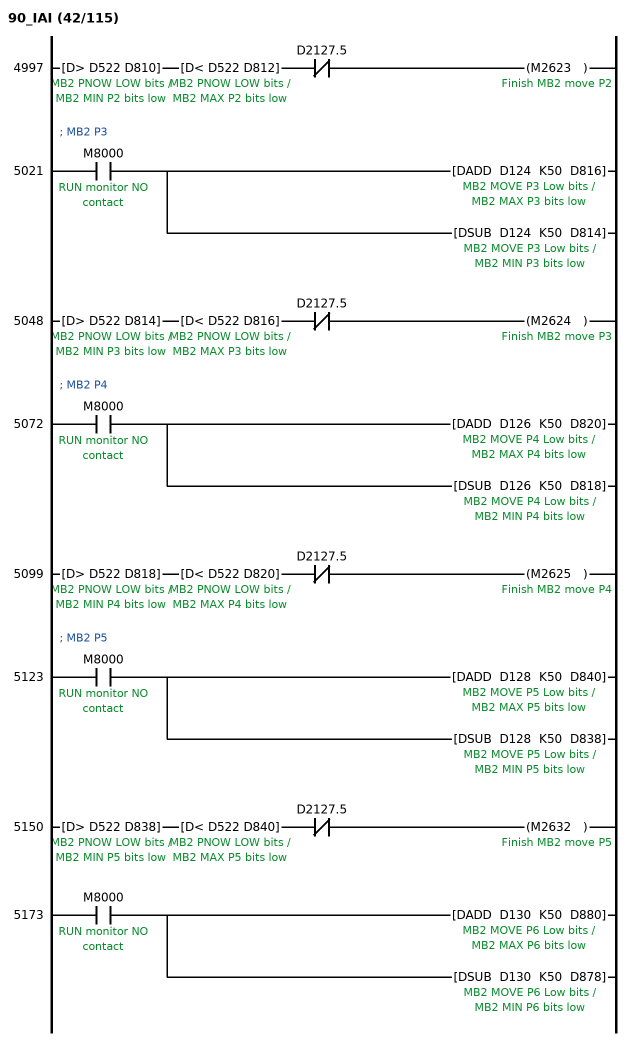
[picture p144: ladder of 90_IAI, rungs at steps 4997 to 5173]
4997  LDD>    D522 D810  ; MB2 PNOW LOW bits / MB2 MIN P2 bits low
      ANDD<   D522 D812  ; MB2 PNOW LOW bits / MB2 MAX P2 bits low
      ANI     D2127.5
      OUT     M2623  ; Finish MB2 move P2
; MB2 P3
5021  LD      M8000  ; RUN monitor NO contact
      DADD    D124 K50 D816  ; MB2 MAX P3 bits low
      DSUB    D124 K50 D814  ; MB2 MIN P3 bits low
5048  LDD>    D522 D814  ; MB2 PNOW LOW bits / MB2 MIN P3 bits low
      ANDD<   D522 D816  ; MB2 PNOW LOW bits / MB2 MAX P3 bits low
      ANI     D2127.5
      OUT     M2624  ; Finish MB2 move P3
; MB2 P4
5072  LD      M8000  ; RUN monitor NO contact
      DADD    D126 K50 D820  ; MB2 MAX P4 bits low
      DSUB    D126 K50 D818  ; MB2 MIN P4 bits low
5099  LDD>    D522 D818  ; MB2 PNOW LOW bits / MB2 MIN P4 bits low
      ANDD<   D522 D820  ; MB2 PNOW LOW bits / MB2 MAX P4 bits low
      ANI     D2127.5
      OUT     M2625  ; Finish MB2 move P4
; MB2 P5
5123  LD      M8000  ; RUN monitor NO contact
      DADD    D128 K50 D840  ; MB2 MAX P5 bits low
      DSUB    D128 K50 D838  ; MB2 MIN P5 bits low
5150  LDD>    D522 D838  ; MB2 PNOW LOW bits / MB2 MIN P5 bits low
      ANDD<   D522 D840  ; MB2 PNOW LOW bits / MB2 MAX P5 bits low
      ANI     D2127.5
      OUT     M2632  ; Finish MB2 move P5
5173  LD      M8000  ; RUN monitor NO contact
      DADD    D130 K50 D880  ; MB2 MAX P6 bits low
      DSUB    D130 K50 D878  ; MB2 MIN P6 bits low
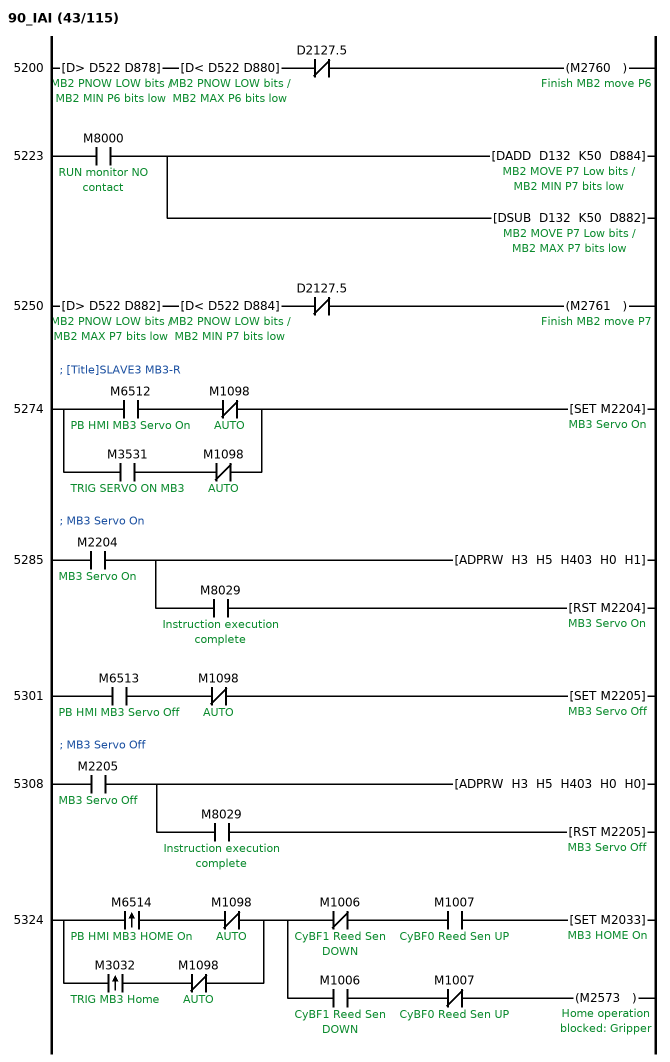
5200  LDD>    D522 D878  ; MB2 PNOW LOW bits / MB2 MIN P6 bits low
      ANDD<   D522 D880  ; MB2 PNOW LOW bits / MB2 MAX P6 bits low
      ANI     D2127.5
      OUT     M2760  ; Finish MB2 move P6
5223  LD      M8000  ; RUN monitor NO contact
      DADD    D132 K50 D884  ; MB2 MIN P7 bits low
      DSUB    D132 K50 D882  ; MB2 MAX P7 bits low
5250  LDD>    D522 D882  ; MB2 PNOW LOW bits / MB2 MAX P7 bits low
      ANDD<   D522 D884  ; MB2 PNOW LOW bits / MB2 MIN P7 bits low
      ANI     D2127.5
      OUT     M2761  ; Finish MB2 move P7
; [Title]SLAVE3 MB3-R
5274  LD      M6512  ; PB HMI MB3 Servo On
      ANI     M1098  ; AUTO
      LD      M3531  ; TRIG SERVO ON MB3
      ANI     M1098  ; AUTO
      ORB
      SET     M2204  ; MB3 Servo On
; MB3 Servo On
5285  LD      M2204  ; MB3 Servo On
      ADPRW   H3 H5 H403 H0 H1
      AND     M8029  ; Instruction execution complete
      RST     M2204  ; MB3 Servo On
5301  LD      M6513  ; PB HMI MB3 Servo Off
      ANI     M1098  ; AUTO
      SET     M2205  ; MB3 Servo Off
; MB3 Servo Off
5308  LD      M2205  ; MB3 Servo Off
      ADPRW   H3 H5 H403 H0 H0
      AND     M8029  ; Instruction execution complete
      RST     M2205  ; MB3 Servo Off
5324  LDP     M6514  ; PB HMI MB3 HOME On
      ANI     M1098  ; AUTO
      LDP     M3032  ; TRIG MB3 Home
      ANI     M1098  ; AUTO
      ORB
      MPS
      ANI     M1006  ; CyBF1 Reed Sen DOWN
      AND     M1007  ; CyBF0 Reed Sen UP
      SET     M2033  ; MB3 HOME On
      MPP
      AND     M1006  ; CyBF1 Reed Sen DOWN
      ANI     M1007  ; CyBF0 Reed Sen UP
      OUT     M2573  ; Home operation blocked: Gripper
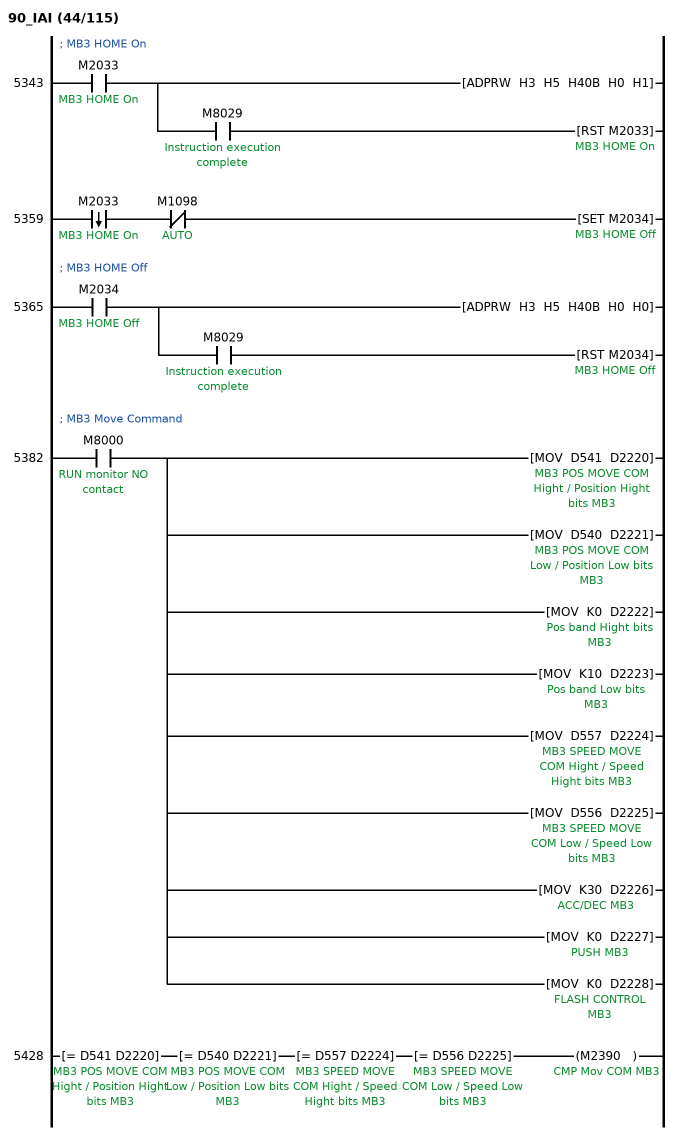
; MB3 HOME On
5343  LD      M2033  ; MB3 HOME On
      ADPRW   H3 H5 H40B H0 H1
      AND     M8029  ; Instruction execution complete
      RST     M2033  ; MB3 HOME On
5359  LDF     M2033  ; MB3 HOME On
      ANI     M1098  ; AUTO
      SET     M2034  ; MB3 HOME Off
; MB3 HOME Off
5365  LD      M2034  ; MB3 HOME Off
      ADPRW   H3 H5 H40B H0 H0
      AND     M8029  ; Instruction execution complete
      RST     M2034  ; MB3 HOME Off
; MB3 Move Command
5382  LD      M8000  ; RUN monitor NO contact
      MOV     D541 D2220  ; MB3 POS MOVE COM Hight / Position Hight bits MB3
      MOV     D540 D2221  ; MB3 POS MOVE COM Low / Position Low bits MB3
      MOV     K0 D2222  ; Pos band Hight bits MB3
      MOV     K10 D2223  ; Pos band Low bits MB3
      MOV     D557 D2224  ; MB3 SPEED MOVE COM Hight / Speed Hight bits MB3
      MOV     D556 D2225  ; MB3 SPEED MOVE COM Low / Speed Low bits MB3
      MOV     K30 D2226  ; ACC/DEC MB3
      MOV     K0 D2227  ; PUSH MB3
      MOV     K0 D2228  ; FLASH CONTROL MB3
5428  LD=     D541 D2220  ; MB3 POS MOVE COM Hight / Position Hight bits MB3
      AND=    D540 D2221  ; MB3 POS MOVE COM Low / Position Low bits MB3
      AND=    D557 D2224  ; MB3 SPEED MOVE COM Hight / Speed Hight bits MB3
      AND=    D556 D2225  ; MB3 SPEED MOVE COM Low / Speed Low bits MB3
      OUT     M2390  ; CMP Mov COM MB3
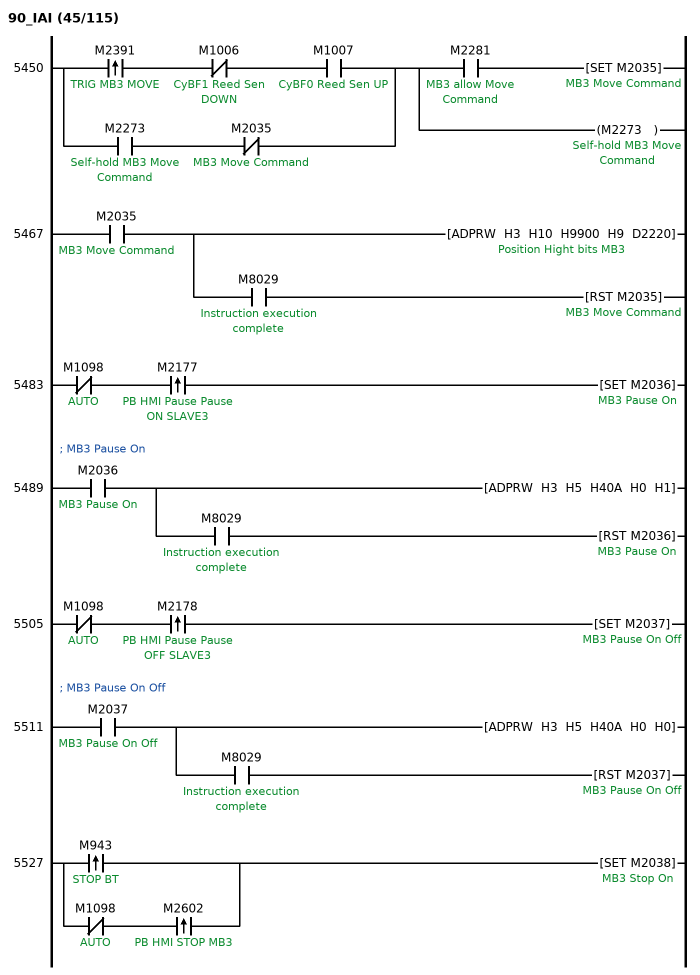
5450  LDP     M2391  ; TRIG MB3 MOVE
      ANI     M1006  ; CyBF1 Reed Sen DOWN
      AND     M1007  ; CyBF0 Reed Sen UP
      LD      M2273  ; Self-hold MB3 Move Command
      ANI     M2035  ; MB3 Move Command
      ORB
      MPS
      AND     M2281  ; MB3 allow Move Command
      SET     M2035  ; MB3 Move Command
      MPP
      OUT     M2273  ; Self-hold MB3 Move Command
5467  LD      M2035  ; MB3 Move Command
      ADPRW   H3 H10 H9900 H9 D2220
      AND     M8029  ; Instruction execution complete
      RST     M2035  ; MB3 Move Command
5483  LDI     M1098  ; AUTO
      ANDP    M2177  ; PB HMI Pause Pause ON SLAVE3
      SET     M2036  ; MB3 Pause On
; MB3 Pause On
5489  LD      M2036  ; MB3 Pause On
      ADPRW   H3 H5 H40A H0 H1
      AND     M8029  ; Instruction execution complete
      RST     M2036  ; MB3 Pause On
5505  LDI     M1098  ; AUTO
      ANDP    M2178  ; PB HMI Pause Pause OFF SLAVE3
      SET     M2037  ; MB3 Pause On Off
; MB3 Pause On Off
5511  LD      M2037  ; MB3 Pause On Off
      ADPRW   H3 H5 H40A H0 H0
      AND     M8029  ; Instruction execution complete
      RST     M2037  ; MB3 Pause On Off
5527  LDP     M943  ; STOP BT
      LDI     M1098  ; AUTO
      ANDP    M2602  ; PB HMI STOP MB3
      ORB
      SET     M2038  ; MB3 Stop On
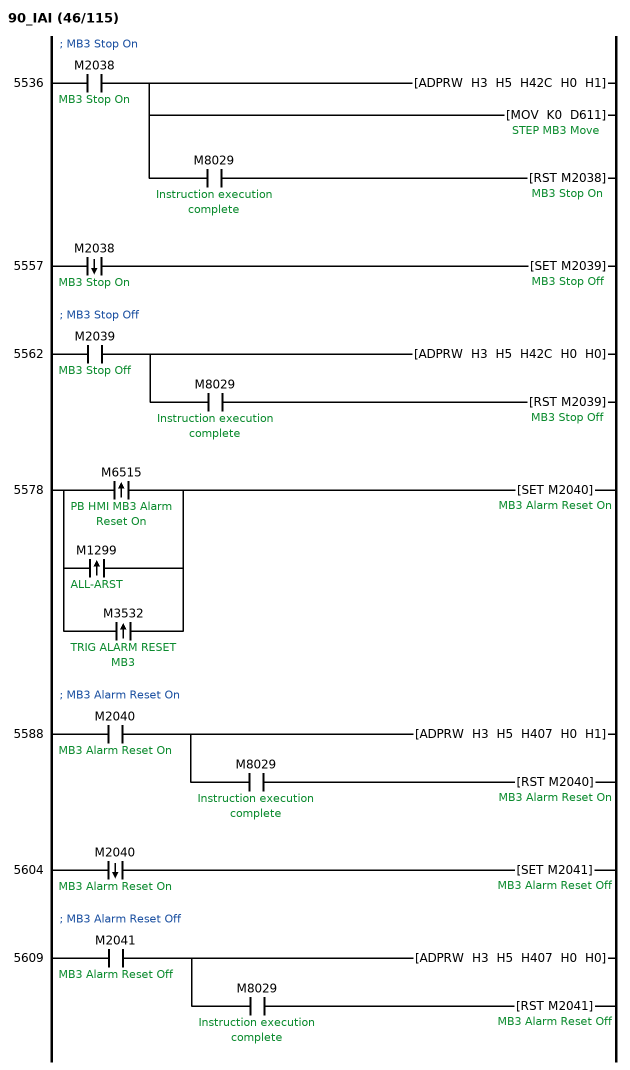
; MB3 Stop On
5536  LD      M2038  ; MB3 Stop On
      ADPRW   H3 H5 H42C H0 H1
      MOV     K0 D611  ; STEP MB3 Move
      AND     M8029  ; Instruction execution complete
      RST     M2038  ; MB3 Stop On
5557  LDF     M2038  ; MB3 Stop On
      SET     M2039  ; MB3 Stop Off
; MB3 Stop Off
5562  LD      M2039  ; MB3 Stop Off
      ADPRW   H3 H5 H42C H0 H0
      AND     M8029  ; Instruction execution complete
      RST     M2039  ; MB3 Stop Off
5578  LDP     M6515  ; PB HMI MB3 Alarm Reset On
      ORP     M1299  ; ALL-ARST
      ORP     M3532  ; TRIG ALARM RESET MB3
      SET     M2040  ; MB3 Alarm Reset On
; MB3 Alarm Reset On
5588  LD      M2040  ; MB3 Alarm Reset On
      ADPRW   H3 H5 H407 H0 H1
      AND     M8029  ; Instruction execution complete
      RST     M2040  ; MB3 Alarm Reset On
5604  LDF     M2040  ; MB3 Alarm Reset On
      SET     M2041  ; MB3 Alarm Reset Off
; MB3 Alarm Reset Off
5609  LD      M2041  ; MB3 Alarm Reset Off
      ADPRW   H3 H5 H407 H0 H0
      AND     M8029  ; Instruction execution complete
      RST     M2041  ; MB3 Alarm Reset Off
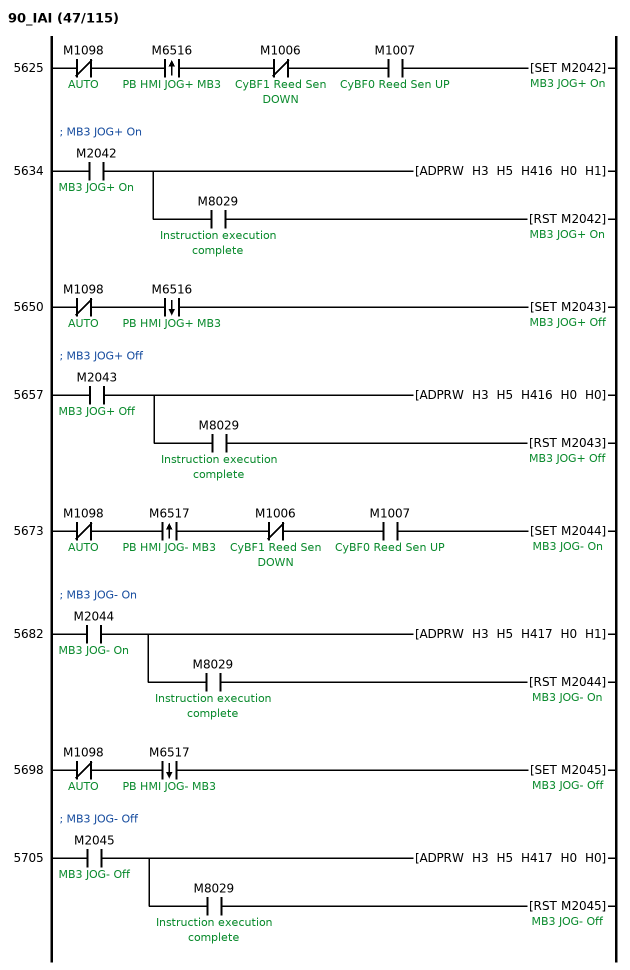
5625  LDI     M1098  ; AUTO
      ANDP    M6516  ; PB HMI JOG+ MB3
      ANI     M1006  ; CyBF1 Reed Sen DOWN
      AND     M1007  ; CyBF0 Reed Sen UP
      SET     M2042  ; MB3 JOG+ On
; MB3 JOG+ On
5634  LD      M2042  ; MB3 JOG+ On
      ADPRW   H3 H5 H416 H0 H1
      AND     M8029  ; Instruction execution complete
      RST     M2042  ; MB3 JOG+ On
5650  LDI     M1098  ; AUTO
      ANDF    M6516  ; PB HMI JOG+ MB3
      SET     M2043  ; MB3 JOG+ Off
; MB3 JOG+ Off
5657  LD      M2043  ; MB3 JOG+ Off
      ADPRW   H3 H5 H416 H0 H0
      AND     M8029  ; Instruction execution complete
      RST     M2043  ; MB3 JOG+ Off
5673  LDI     M1098  ; AUTO
      ANDP    M6517  ; PB HMI JOG- MB3
      ANI     M1006  ; CyBF1 Reed Sen DOWN
      AND     M1007  ; CyBF0 Reed Sen UP
      SET     M2044  ; MB3 JOG- On
; MB3 JOG- On
5682  LD      M2044  ; MB3 JOG- On
      ADPRW   H3 H5 H417 H0 H1
      AND     M8029  ; Instruction execution complete
      RST     M2044  ; MB3 JOG- On
5698  LDI     M1098  ; AUTO
      ANDF    M6517  ; PB HMI JOG- MB3
      SET     M2045  ; MB3 JOG- Off
; MB3 JOG- Off
5705  LD      M2045  ; MB3 JOG- Off
      ADPRW   H3 H5 H417 H0 H0
      AND     M8029  ; Instruction execution complete
      RST     M2045  ; MB3 JOG- Off
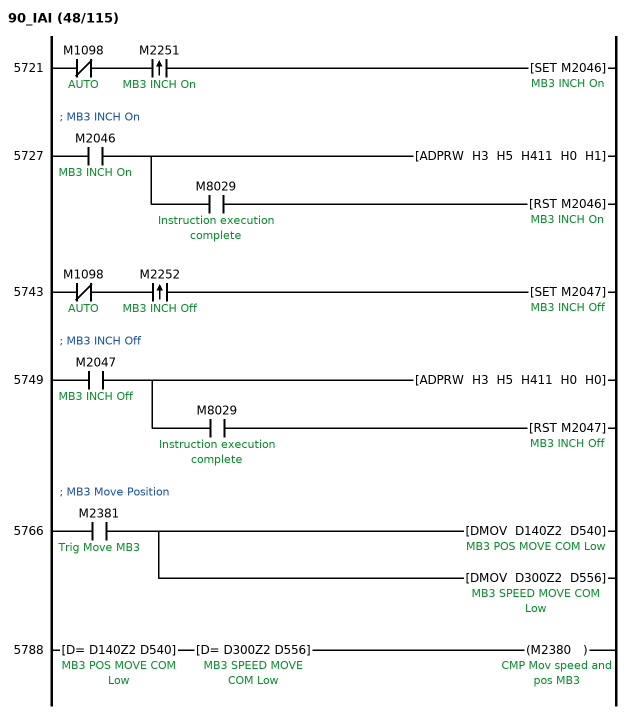
5721  LDI     M1098  ; AUTO
      ANDP    M2251  ; MB3 INCH On
      SET     M2046  ; MB3 INCH On
; MB3 INCH On
5727  LD      M2046  ; MB3 INCH On
      ADPRW   H3 H5 H411 H0 H1
      AND     M8029  ; Instruction execution complete
      RST     M2046  ; MB3 INCH On
5743  LDI     M1098  ; AUTO
      ANDP    M2252  ; MB3 INCH Off
      SET     M2047  ; MB3 INCH Off
; MB3 INCH Off
5749  LD      M2047  ; MB3 INCH Off
      ADPRW   H3 H5 H411 H0 H0
      AND     M8029  ; Instruction execution complete
      RST     M2047  ; MB3 INCH Off
; MB3 Move Position
5766  LD      M2381  ; Trig Move MB3
      DMOV    D140Z2 D540
        [note] Position
      DMOV    D300Z2 D556
        [note] Speed
5788  LDD=    D140Z2 D540  ; MB3 POS MOVE COM Low
      ANDD=   D300Z2 D556  ; MB3 SPEED MOVE COM Low
      OUT     M2380  ; CMP Mov speed and pos MB3
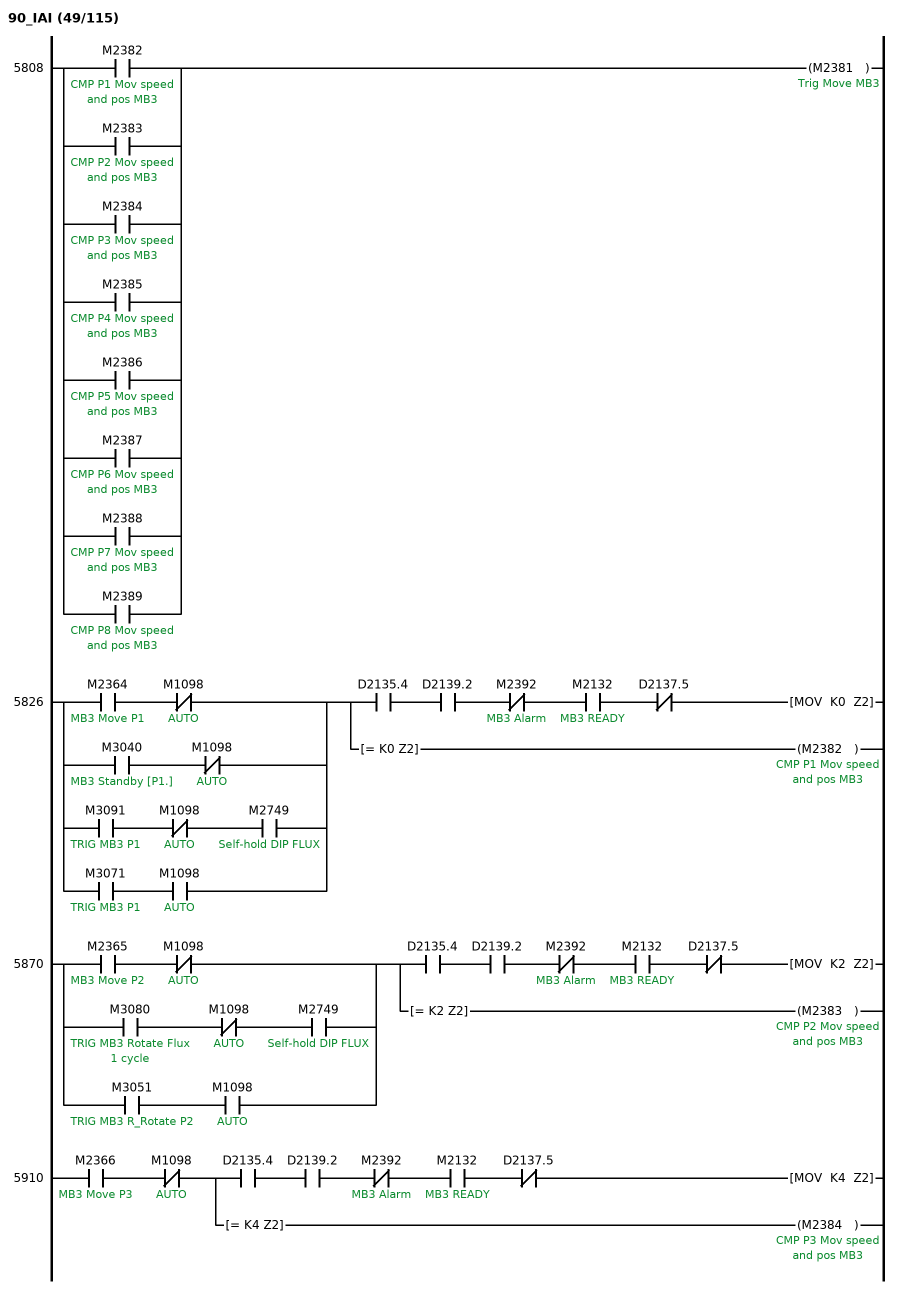
5808  LD      M2382  ; CMP P1 Mov speed and pos MB3
      OR      M2383  ; CMP P2 Mov speed and pos MB3
      OR      M2384  ; CMP P3 Mov speed and pos MB3
      OR      M2385  ; CMP P4 Mov speed and pos MB3
      OR      M2386  ; CMP P5 Mov speed and pos MB3
      OR      M2387  ; CMP P6 Mov speed and pos MB3
      OR      M2388  ; CMP P7 Mov speed and pos MB3
      OR      M2389  ; CMP P8 Mov speed and pos MB3
      OUT     M2381  ; Trig Move MB3
5826  LD      M2364  ; MB3 Move P1
      ANI     M1098  ; AUTO
      LD      M3040  ; MB3 Standby [P1.]
      ANI     M1098  ; AUTO
      ORB
      LD      M3091  ; TRIG MB3 P1
      ANI     M1098  ; AUTO
      AND     M2749  ; Self-hold DIP FLUX
      ORB
      LD      M3071  ; TRIG MB3 P1
      AND     M1098  ; AUTO
      ORB
      MPS
      AND     D2135.4
      AND     D2139.2
      ANI     M2392  ; MB3 Alarm
      AND     M2132  ; MB3 READY
      ANI     D2137.5
      MOV     K0 Z2
      MPP
      AND=    K0 Z2
      OUT     M2382  ; CMP P1 Mov speed and pos MB3
5870  LD      M2365  ; MB3 Move P2
      ANI     M1098  ; AUTO
      LD      M3080  ; TRIG MB3 Rotate Flux 1 cycle
      ANI     M1098  ; AUTO
      AND     M2749  ; Self-hold DIP FLUX
      ORB
      LD      M3051  ; TRIG MB3 R_Rotate P2
      AND     M1098  ; AUTO
      ORB
      MPS
      AND     D2135.4
      AND     D2139.2
      ANI     M2392  ; MB3 Alarm
      AND     M2132  ; MB3 READY
      ANI     D2137.5
      MOV     K2 Z2
      MPP
      AND=    K2 Z2
      OUT     M2383  ; CMP P2 Mov speed and pos MB3
5910  LD      M2366  ; MB3 Move P3
      ANI     M1098  ; AUTO
      MPS
      AND     D2135.4
      AND     D2139.2
      ANI     M2392  ; MB3 Alarm
      AND     M2132  ; MB3 READY
      ANI     D2137.5
      MOV     K4 Z2
      MPP
      AND=    K4 Z2
      OUT     M2384  ; CMP P3 Mov speed and pos MB3
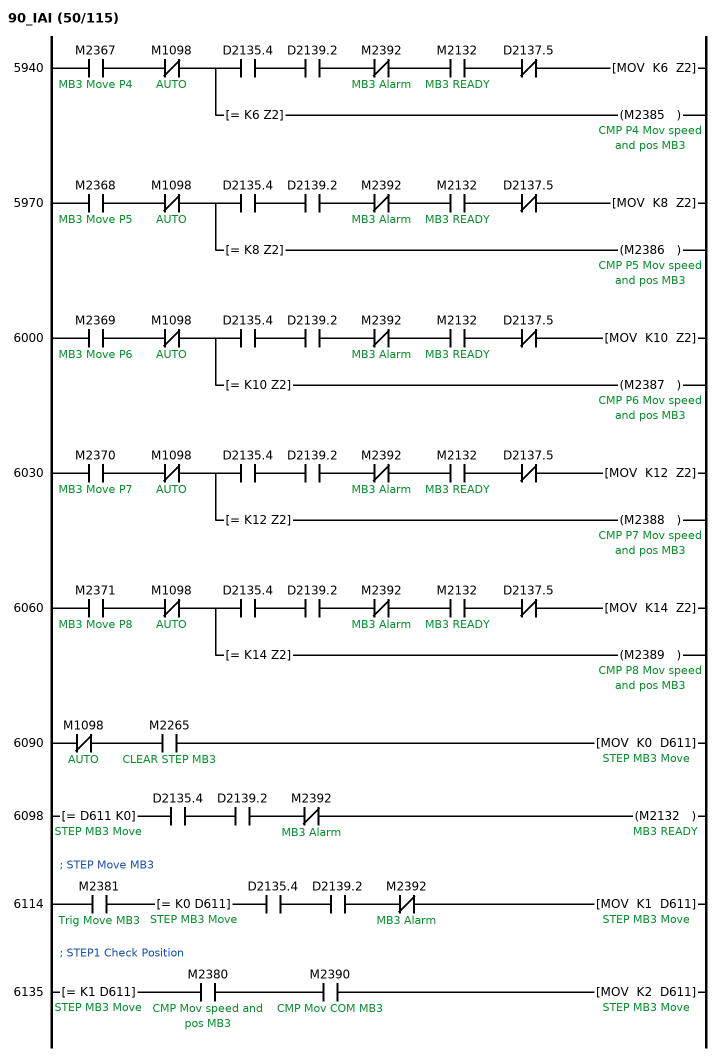
5940  LD      M2367  ; MB3 Move P4
      ANI     M1098  ; AUTO
      MPS
      AND     D2135.4
      AND     D2139.2
      ANI     M2392  ; MB3 Alarm
      AND     M2132  ; MB3 READY
      ANI     D2137.5
      MOV     K6 Z2
      MPP
      AND=    K6 Z2
      OUT     M2385  ; CMP P4 Mov speed and pos MB3
5970  LD      M2368  ; MB3 Move P5
      ANI     M1098  ; AUTO
      MPS
      AND     D2135.4
      AND     D2139.2
      ANI     M2392  ; MB3 Alarm
      AND     M2132  ; MB3 READY
      ANI     D2137.5
      MOV     K8 Z2
      MPP
      AND=    K8 Z2
      OUT     M2386  ; CMP P5 Mov speed and pos MB3
6000  LD      M2369  ; MB3 Move P6
      ANI     M1098  ; AUTO
      MPS
      AND     D2135.4
      AND     D2139.2
      ANI     M2392  ; MB3 Alarm
      AND     M2132  ; MB3 READY
      ANI     D2137.5
      MOV     K10 Z2
      MPP
      AND=    K10 Z2
      OUT     M2387  ; CMP P6 Mov speed and pos MB3
6030  LD      M2370  ; MB3 Move P7
      ANI     M1098  ; AUTO
      MPS
      AND     D2135.4
      AND     D2139.2
      ANI     M2392  ; MB3 Alarm
      AND     M2132  ; MB3 READY
      ANI     D2137.5
      MOV     K12 Z2
      MPP
      AND=    K12 Z2
      OUT     M2388  ; CMP P7 Mov speed and pos MB3
6060  LD      M2371  ; MB3 Move P8
      ANI     M1098  ; AUTO
      MPS
      AND     D2135.4
      AND     D2139.2
      ANI     M2392  ; MB3 Alarm
      AND     M2132  ; MB3 READY
      ANI     D2137.5
      MOV     K14 Z2
      MPP
      AND=    K14 Z2
      OUT     M2389  ; CMP P8 Mov speed and pos MB3
6090  LDI     M1098  ; AUTO
      AND     M2265  ; CLEAR STEP MB3
      MOV     K0 D611
6098  LD=     D611 K0  ; STEP MB3 Move
      AND     D2135.4
      AND     D2139.2
      ANI     M2392  ; MB3 Alarm
      OUT     M2132  ; MB3 READY
; STEP Move MB3
6114  LD      M2381  ; Trig Move MB3
      AND=    K0 D611  ; STEP MB3 Move
      AND     D2135.4
      AND     D2139.2
      ANI     M2392  ; MB3 Alarm
      MOV     K1 D611
; STEP1 Check Position
6135  LD=     K1 D611  ; STEP MB3 Move
      AND     M2380  ; CMP Mov speed and pos MB3
      AND     M2390  ; CMP Mov COM MB3
      MOV     K2 D611
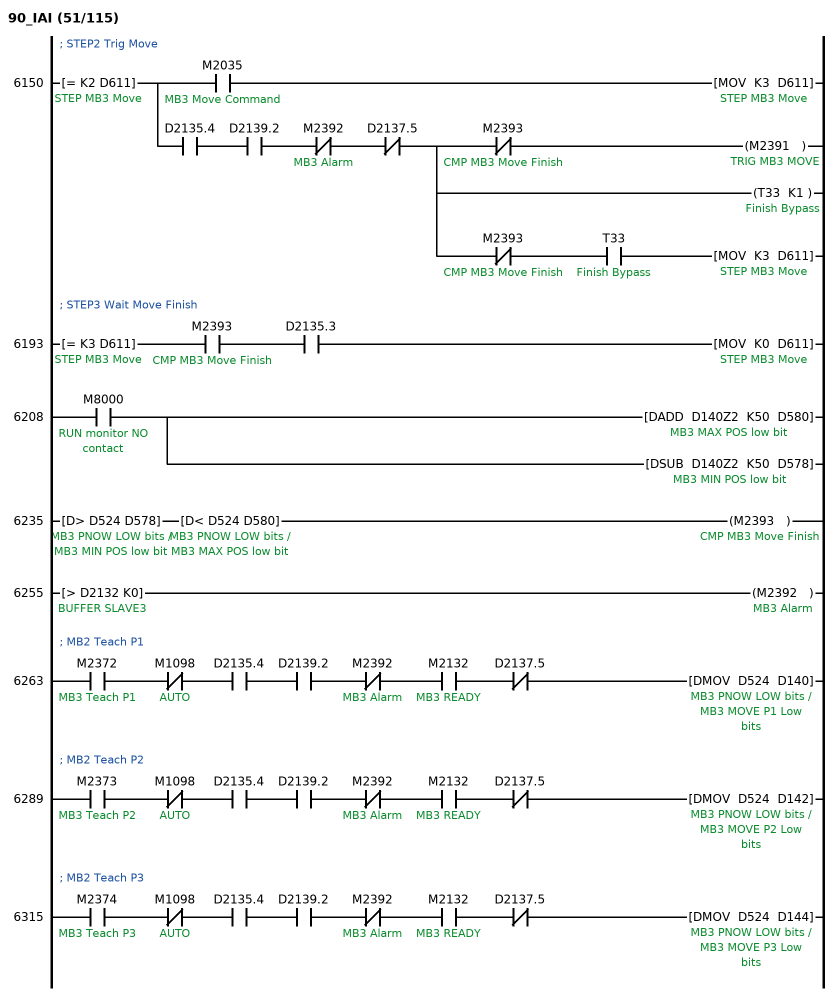
; STEP2 Trig Move
6150  LD=     K2 D611  ; STEP MB3 Move
      MPS
      AND     M2035  ; MB3 Move Command
      MOV     K3 D611
      MPP
      AND     D2135.4
      AND     D2139.2
      ANI     M2392  ; MB3 Alarm
      ANI     D2137.5
      MPS
      ANI     M2393  ; CMP MB3 Move Finish
      OUT     M2391  ; TRIG MB3 MOVE
      MPP
      OUT     T33 K1  ; Finish Bypass
      ANI     M2393  ; CMP MB3 Move Finish
      AND     T33  ; Finish Bypass
      MOV     K3 D611
; STEP3 Wait Move Finish
6193  LD=     K3 D611  ; STEP MB3 Move
      AND     M2393  ; CMP MB3 Move Finish
      AND     D2135.3
      MOV     K0 D611
6208  LD      M8000  ; RUN monitor NO contact
      DADD    D140Z2 K50 D580  ; MB3 MAX POS low bit
      DSUB    D140Z2 K50 D578  ; MB3 MIN POS low bit
6235  LDD>    D524 D578  ; MB3 PNOW LOW bits / MB3 MIN POS low bit
      ANDD<   D524 D580  ; MB3 PNOW LOW bits / MB3 MAX POS low bit
      OUT     M2393  ; CMP MB3 Move Finish
6255  LD>     D2132 K0  ; BUFFER SLAVE3
      OUT     M2392  ; MB3 Alarm
; MB2 Teach P1
6263  LD      M2372  ; MB3 Teach P1
      ANI     M1098  ; AUTO
      AND     D2135.4
      AND     D2139.2
      ANI     M2392  ; MB3 Alarm
      AND     M2132  ; MB3 READY
      ANI     D2137.5
      DMOV    D524 D140  ; MB3 MOVE P1 Low bits
; MB2 Teach P2
6289  LD      M2373  ; MB3 Teach P2
      ANI     M1098  ; AUTO
      AND     D2135.4
      AND     D2139.2
      ANI     M2392  ; MB3 Alarm
      AND     M2132  ; MB3 READY
      ANI     D2137.5
      DMOV    D524 D142  ; MB3 MOVE P2 Low bits
; MB2 Teach P3
6315  LD      M2374  ; MB3 Teach P3
      ANI     M1098  ; AUTO
      AND     D2135.4
      AND     D2139.2
      ANI     M2392  ; MB3 Alarm
      AND     M2132  ; MB3 READY
      ANI     D2137.5
      DMOV    D524 D144  ; MB3 MOVE P3 Low bits
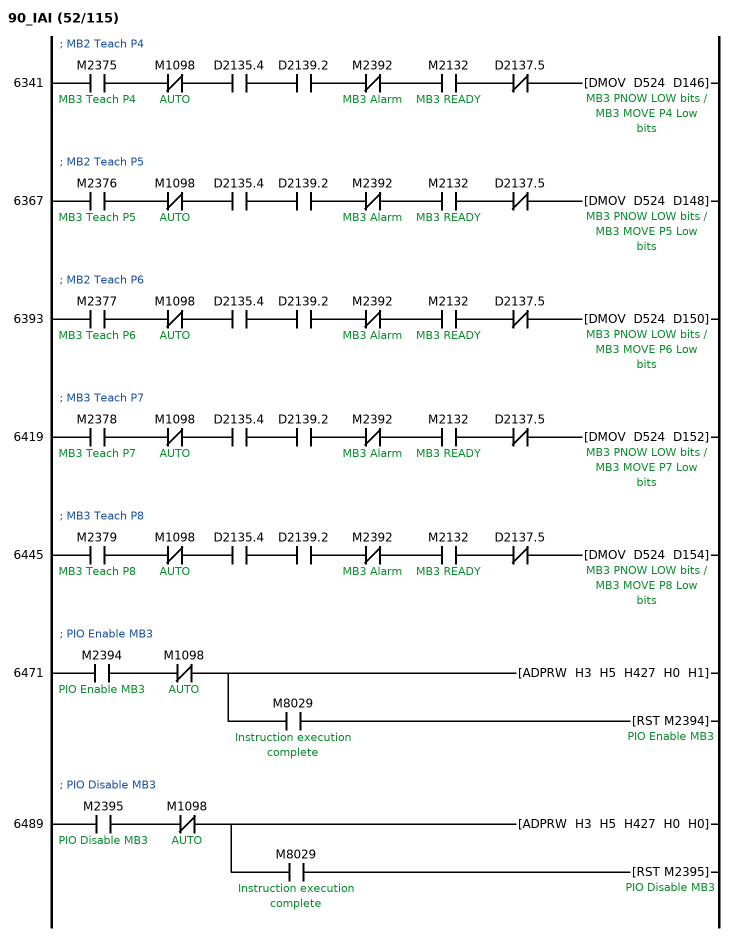
; MB2 Teach P4
6341  LD      M2375  ; MB3 Teach P4
      ANI     M1098  ; AUTO
      AND     D2135.4
      AND     D2139.2
      ANI     M2392  ; MB3 Alarm
      AND     M2132  ; MB3 READY
      ANI     D2137.5
      DMOV    D524 D146  ; MB3 MOVE P4 Low bits
; MB2 Teach P5
6367  LD      M2376  ; MB3 Teach P5
      ANI     M1098  ; AUTO
      AND     D2135.4
      AND     D2139.2
      ANI     M2392  ; MB3 Alarm
      AND     M2132  ; MB3 READY
      ANI     D2137.5
      DMOV    D524 D148  ; MB3 MOVE P5 Low bits
; MB2 Teach P6
6393  LD      M2377  ; MB3 Teach P6
      ANI     M1098  ; AUTO
      AND     D2135.4
      AND     D2139.2
      ANI     M2392  ; MB3 Alarm
      AND     M2132  ; MB3 READY
      ANI     D2137.5
      DMOV    D524 D150  ; MB3 MOVE P6 Low bits
; MB3 Teach P7
6419  LD      M2378  ; MB3 Teach P7
      ANI     M1098  ; AUTO
      AND     D2135.4
      AND     D2139.2
      ANI     M2392  ; MB3 Alarm
      AND     M2132  ; MB3 READY
      ANI     D2137.5
      DMOV    D524 D152  ; MB3 MOVE P7 Low bits
; MB3 Teach P8
6445  LD      M2379  ; MB3 Teach P8
      ANI     M1098  ; AUTO
      AND     D2135.4
      AND     D2139.2
      ANI     M2392  ; MB3 Alarm
      AND     M2132  ; MB3 READY
      ANI     D2137.5
      DMOV    D524 D154  ; MB3 MOVE P8 Low bits
; PIO Enable MB3
6471  LD      M2394  ; PIO Enable MB3
      ANI     M1098  ; AUTO
      ADPRW   H3 H5 H427 H0 H1
      AND     M8029  ; Instruction execution complete
      RST     M2394  ; PIO Enable MB3
; PIO Disable MB3
6489  LD      M2395  ; PIO Disable MB3
      ANI     M1098  ; AUTO
      ADPRW   H3 H5 H427 H0 H0
      AND     M8029  ; Instruction execution complete
      RST     M2395  ; PIO Disable MB3
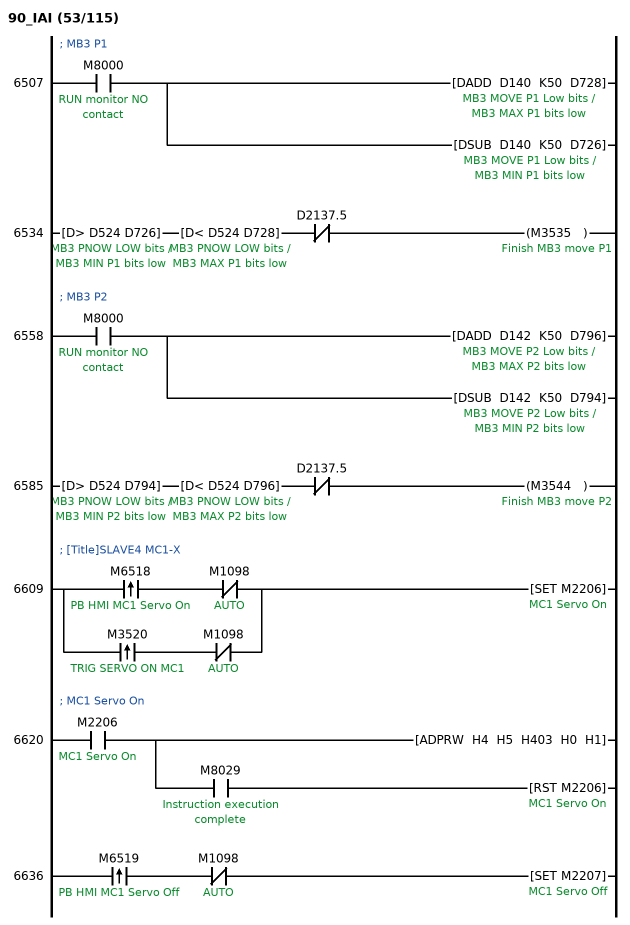
; MB3 P1
6507  LD      M8000  ; RUN monitor NO contact
      DADD    D140 K50 D728  ; MB3 MAX P1 bits low
      DSUB    D140 K50 D726  ; MB3 MIN P1 bits low
6534  LDD>    D524 D726  ; MB3 PNOW LOW bits / MB3 MIN P1 bits low
      ANDD<   D524 D728  ; MB3 PNOW LOW bits / MB3 MAX P1 bits low
      ANI     D2137.5
      OUT     M3535  ; Finish MB3 move P1
; MB3 P2
6558  LD      M8000  ; RUN monitor NO contact
      DADD    D142 K50 D796  ; MB3 MAX P2 bits low
      DSUB    D142 K50 D794  ; MB3 MIN P2 bits low
6585  LDD>    D524 D794  ; MB3 PNOW LOW bits / MB3 MIN P2 bits low
      ANDD<   D524 D796  ; MB3 PNOW LOW bits / MB3 MAX P2 bits low
      ANI     D2137.5
      OUT     M3544  ; Finish MB3 move P2
; [Title]SLAVE4 MC1-X
6609  LDP     M6518  ; PB HMI MC1 Servo On
      ANI     M1098  ; AUTO
      LDP     M3520  ; TRIG SERVO ON MC1
      ANI     M1098  ; AUTO
      ORB
      SET     M2206  ; MC1 Servo On
; MC1 Servo On
6620  LD      M2206  ; MC1 Servo On
      ADPRW   H4 H5 H403 H0 H1
      AND     M8029  ; Instruction execution complete
      RST     M2206  ; MC1 Servo On
6636  LDP     M6519  ; PB HMI MC1 Servo Off
      ANI     M1098  ; AUTO
      SET     M2207  ; MC1 Servo Off
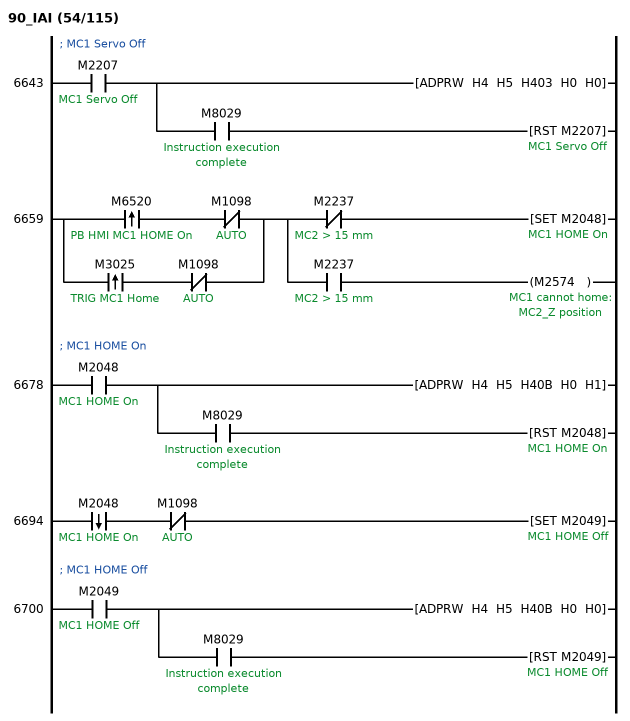
; MC1 Servo Off
6643  LD      M2207  ; MC1 Servo Off
      ADPRW   H4 H5 H403 H0 H0
      AND     M8029  ; Instruction execution complete
      RST     M2207  ; MC1 Servo Off
6659  LDP     M6520  ; PB HMI MC1 HOME On
      ANI     M1098  ; AUTO
      LDP     M3025  ; TRIG MC1 Home
      ANI     M1098  ; AUTO
      ORB
      MPS
      ANI     M2237  ; MC2 > 15 mm
      SET     M2048  ; MC1 HOME On
      MPP
      AND     M2237  ; MC2 > 15 mm
      OUT     M2574  ; MC1 cannot home: MC2_Z position
; MC1 HOME On
6678  LD      M2048  ; MC1 HOME On
      ADPRW   H4 H5 H40B H0 H1
      AND     M8029  ; Instruction execution complete
      RST     M2048  ; MC1 HOME On
6694  LDF     M2048  ; MC1 HOME On
      ANI     M1098  ; AUTO
      SET     M2049  ; MC1 HOME Off
; MC1 HOME Off
6700  LD      M2049  ; MC1 HOME Off
      ADPRW   H4 H5 H40B H0 H0
      AND     M8029  ; Instruction execution complete
      RST     M2049  ; MC1 HOME Off
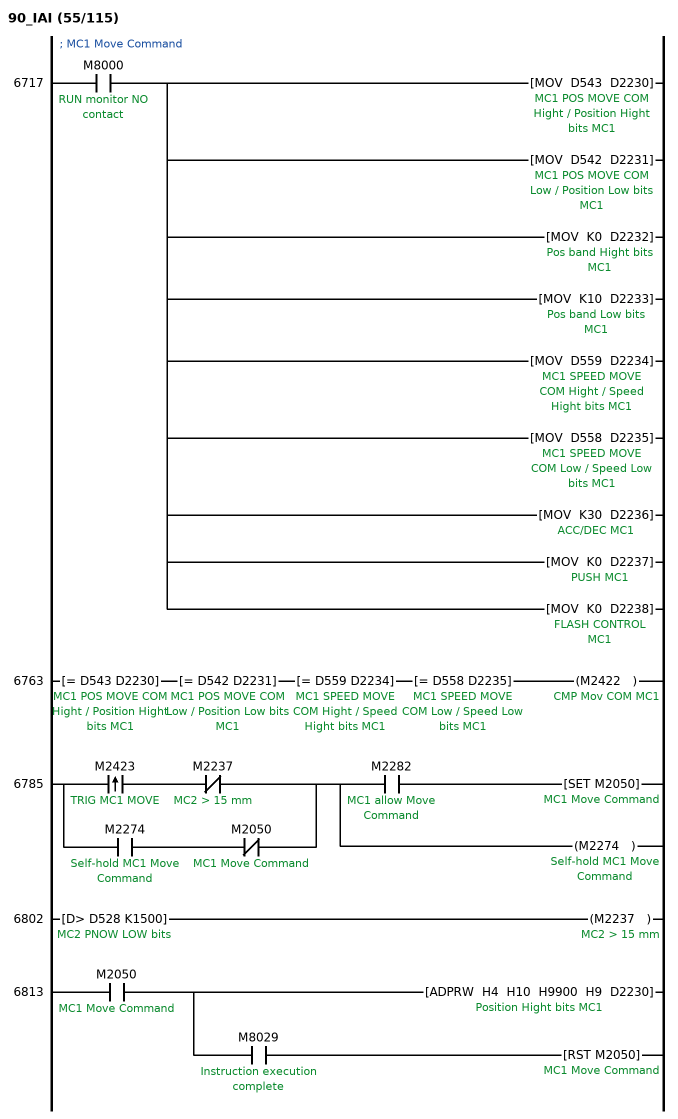
; MC1 Move Command
6717  LD      M8000  ; RUN monitor NO contact
      MOV     D543 D2230  ; MC1 POS MOVE COM Hight / Position Hight bits MC1
      MOV     D542 D2231  ; MC1 POS MOVE COM Low / Position Low bits MC1
      MOV     K0 D2232  ; Pos band Hight bits MC1
      MOV     K10 D2233  ; Pos band Low bits MC1
      MOV     D559 D2234  ; MC1 SPEED MOVE COM Hight / Speed Hight bits MC1
      MOV     D558 D2235  ; MC1 SPEED MOVE COM Low / Speed Low bits MC1
      MOV     K30 D2236  ; ACC/DEC MC1
      MOV     K0 D2237  ; PUSH MC1
      MOV     K0 D2238  ; FLASH CONTROL MC1
6763  LD=     D543 D2230  ; MC1 POS MOVE COM Hight / Position Hight bits MC1
      AND=    D542 D2231  ; MC1 POS MOVE COM Low / Position Low bits MC1
      AND=    D559 D2234  ; MC1 SPEED MOVE COM Hight / Speed Hight bits MC1
      AND=    D558 D2235  ; MC1 SPEED MOVE COM Low / Speed Low bits MC1
      OUT     M2422  ; CMP Mov COM MC1
6785  LDP     M2423  ; TRIG MC1 MOVE
      ANI     M2237  ; MC2 > 15 mm
      LD      M2274  ; Self-hold MC1 Move Command
      ANI     M2050  ; MC1 Move Command
      ORB
      MPS
      AND     M2282  ; MC1 allow Move Command
      SET     M2050  ; MC1 Move Command
      MPP
      OUT     M2274  ; Self-hold MC1 Move Command
6802  LDD>    D528 K1500  ; MC2 PNOW LOW bits
      OUT     M2237  ; MC2 > 15 mm
6813  LD      M2050  ; MC1 Move Command
      ADPRW   H4 H10 H9900 H9 D2230
      AND     M8029  ; Instruction execution complete
      RST     M2050  ; MC1 Move Command
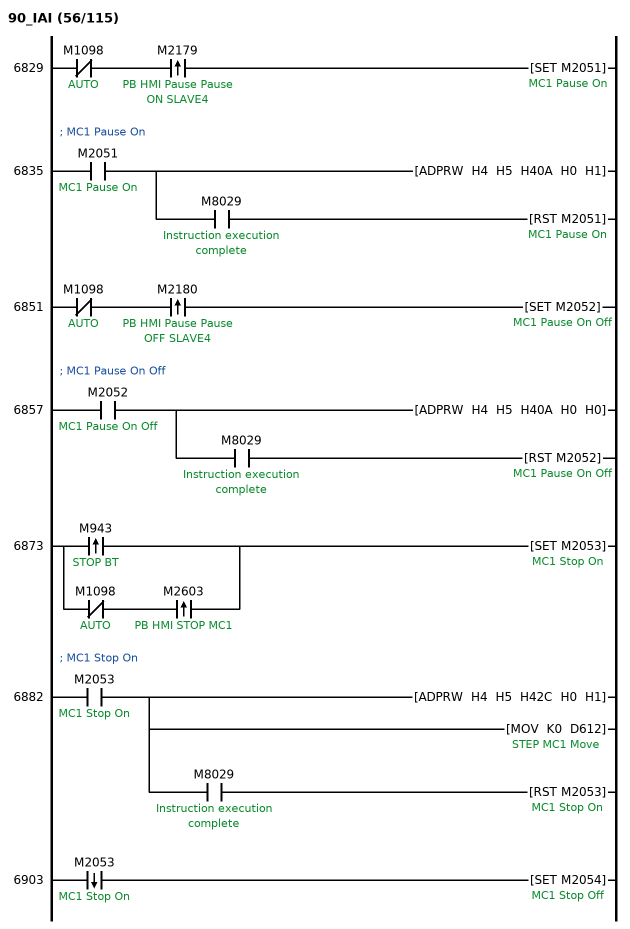
6829  LDI     M1098  ; AUTO
      ANDP    M2179  ; PB HMI Pause Pause ON SLAVE4
      SET     M2051  ; MC1 Pause On
; MC1 Pause On
6835  LD      M2051  ; MC1 Pause On
      ADPRW   H4 H5 H40A H0 H1
      AND     M8029  ; Instruction execution complete
      RST     M2051  ; MC1 Pause On
6851  LDI     M1098  ; AUTO
      ANDP    M2180  ; PB HMI Pause Pause OFF SLAVE4
      SET     M2052  ; MC1 Pause On Off
; MC1 Pause On Off
6857  LD      M2052  ; MC1 Pause On Off
      ADPRW   H4 H5 H40A H0 H0
      AND     M8029  ; Instruction execution complete
      RST     M2052  ; MC1 Pause On Off
6873  LDP     M943  ; STOP BT
      LDI     M1098  ; AUTO
      ANDP    M2603  ; PB HMI STOP MC1
      ORB
      SET     M2053  ; MC1 Stop On
; MC1 Stop On
6882  LD      M2053  ; MC1 Stop On
      ADPRW   H4 H5 H42C H0 H1
      MOV     K0 D612  ; STEP MC1 Move
      AND     M8029  ; Instruction execution complete
      RST     M2053  ; MC1 Stop On
6903  LDF     M2053  ; MC1 Stop On
      SET     M2054  ; MC1 Stop Off
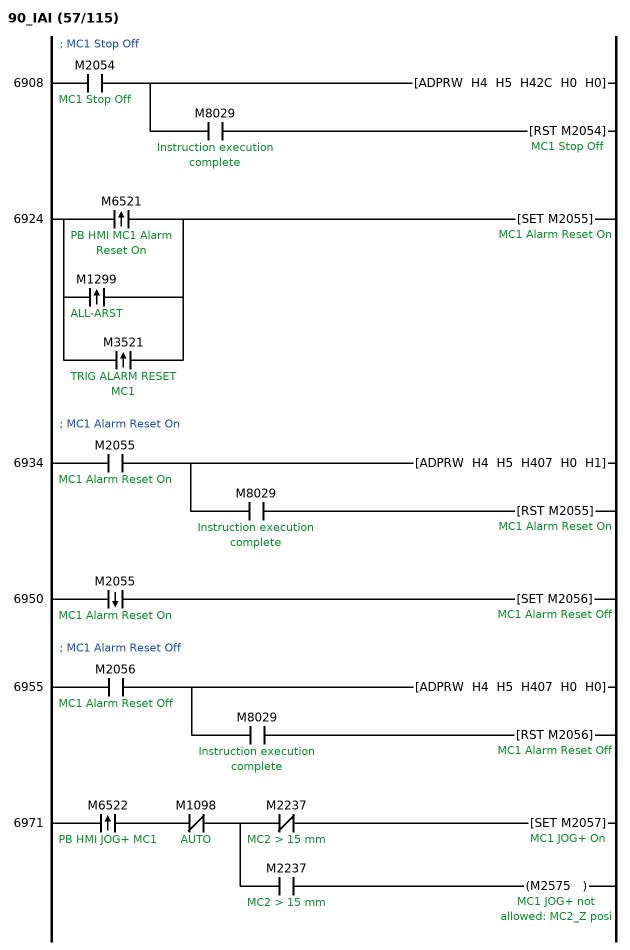
; MC1 Stop Off
6908  LD      M2054  ; MC1 Stop Off
      ADPRW   H4 H5 H42C H0 H0
      AND     M8029  ; Instruction execution complete
      RST     M2054  ; MC1 Stop Off
6924  LDP     M6521  ; PB HMI MC1 Alarm Reset On
      ORP     M1299  ; ALL-ARST
      ORP     M3521  ; TRIG ALARM RESET MC1
      SET     M2055  ; MC1 Alarm Reset On
; MC1 Alarm Reset On
6934  LD      M2055  ; MC1 Alarm Reset On
      ADPRW   H4 H5 H407 H0 H1
      AND     M8029  ; Instruction execution complete
      RST     M2055  ; MC1 Alarm Reset On
6950  LDF     M2055  ; MC1 Alarm Reset On
      SET     M2056  ; MC1 Alarm Reset Off
; MC1 Alarm Reset Off
6955  LD      M2056  ; MC1 Alarm Reset Off
      ADPRW   H4 H5 H407 H0 H0
      AND     M8029  ; Instruction execution complete
      RST     M2056  ; MC1 Alarm Reset Off
6971  LDP     M6522  ; PB HMI JOG+ MC1
      ANI     M1098  ; AUTO
      MPS
      ANI     M2237  ; MC2 > 15 mm
      SET     M2057  ; MC1 JOG+ On
      MPP
      AND     M2237  ; MC2 > 15 mm
      OUT     M2575  ; MC1 JOG+ not allowed: MC2_Z posi
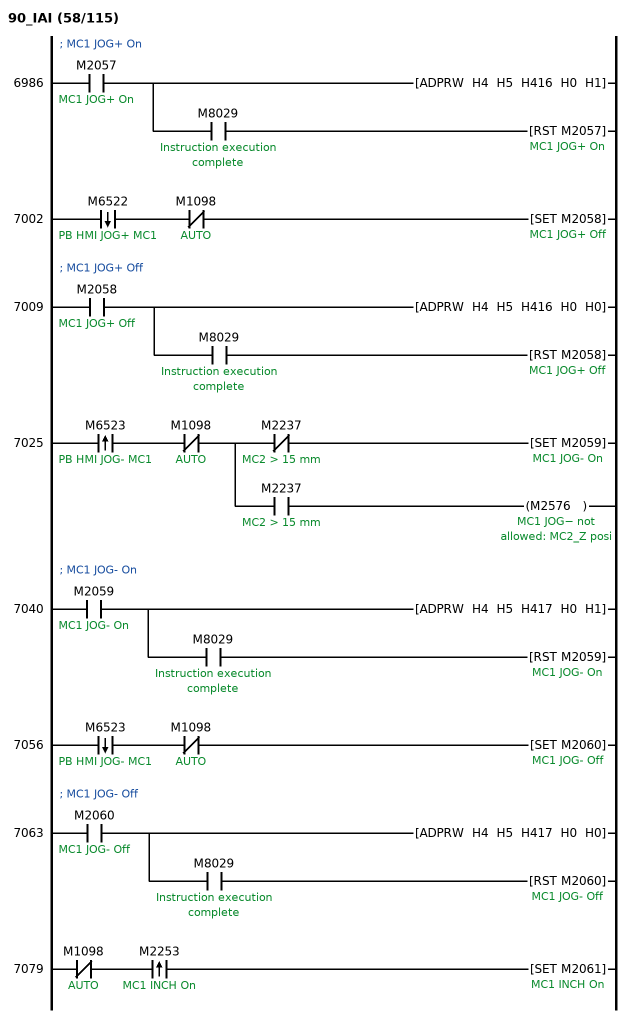
; MC1 JOG+ On
6986  LD      M2057  ; MC1 JOG+ On
      ADPRW   H4 H5 H416 H0 H1
      AND     M8029  ; Instruction execution complete
      RST     M2057  ; MC1 JOG+ On
7002  LDF     M6522  ; PB HMI JOG+ MC1
      ANI     M1098  ; AUTO
      SET     M2058  ; MC1 JOG+ Off
; MC1 JOG+ Off
7009  LD      M2058  ; MC1 JOG+ Off
      ADPRW   H4 H5 H416 H0 H0
      AND     M8029  ; Instruction execution complete
      RST     M2058  ; MC1 JOG+ Off
7025  LDP     M6523  ; PB HMI JOG- MC1
      ANI     M1098  ; AUTO
      MPS
      ANI     M2237  ; MC2 > 15 mm
      SET     M2059  ; MC1 JOG- On
      MPP
      AND     M2237  ; MC2 > 15 mm
      OUT     M2576  ; MC1 JOG− not allowed: MC2_Z posi
; MC1 JOG- On
7040  LD      M2059  ; MC1 JOG- On
      ADPRW   H4 H5 H417 H0 H1
      AND     M8029  ; Instruction execution complete
      RST     M2059  ; MC1 JOG- On
7056  LDF     M6523  ; PB HMI JOG- MC1
      ANI     M1098  ; AUTO
      SET     M2060  ; MC1 JOG- Off
; MC1 JOG- Off
7063  LD      M2060  ; MC1 JOG- Off
      ADPRW   H4 H5 H417 H0 H0
      AND     M8029  ; Instruction execution complete
      RST     M2060  ; MC1 JOG- Off
7079  LDI     M1098  ; AUTO
      ANDP    M2253  ; MC1 INCH On
      SET     M2061  ; MC1 INCH On
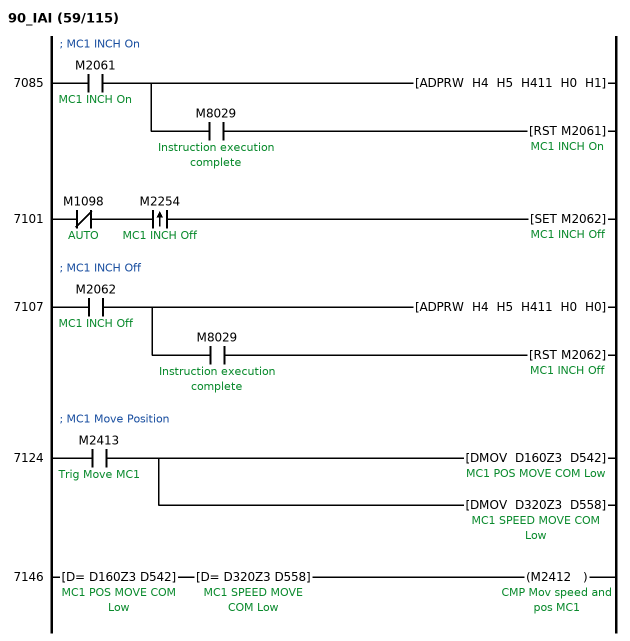
; MC1 INCH On
7085  LD      M2061  ; MC1 INCH On
      ADPRW   H4 H5 H411 H0 H1
      AND     M8029  ; Instruction execution complete
      RST     M2061  ; MC1 INCH On
7101  LDI     M1098  ; AUTO
      ANDP    M2254  ; MC1 INCH Off
      SET     M2062  ; MC1 INCH Off
; MC1 INCH Off
7107  LD      M2062  ; MC1 INCH Off
      ADPRW   H4 H5 H411 H0 H0
      AND     M8029  ; Instruction execution complete
      RST     M2062  ; MC1 INCH Off
; MC1 Move Position
7124  LD      M2413  ; Trig Move MC1
      DMOV    D160Z3 D542
        [note] Position
      DMOV    D320Z3 D558
        [note] Speed
7146  LDD=    D160Z3 D542  ; MC1 POS MOVE COM Low
      ANDD=   D320Z3 D558  ; MC1 SPEED MOVE COM Low
      OUT     M2412  ; CMP Mov speed and pos MC1
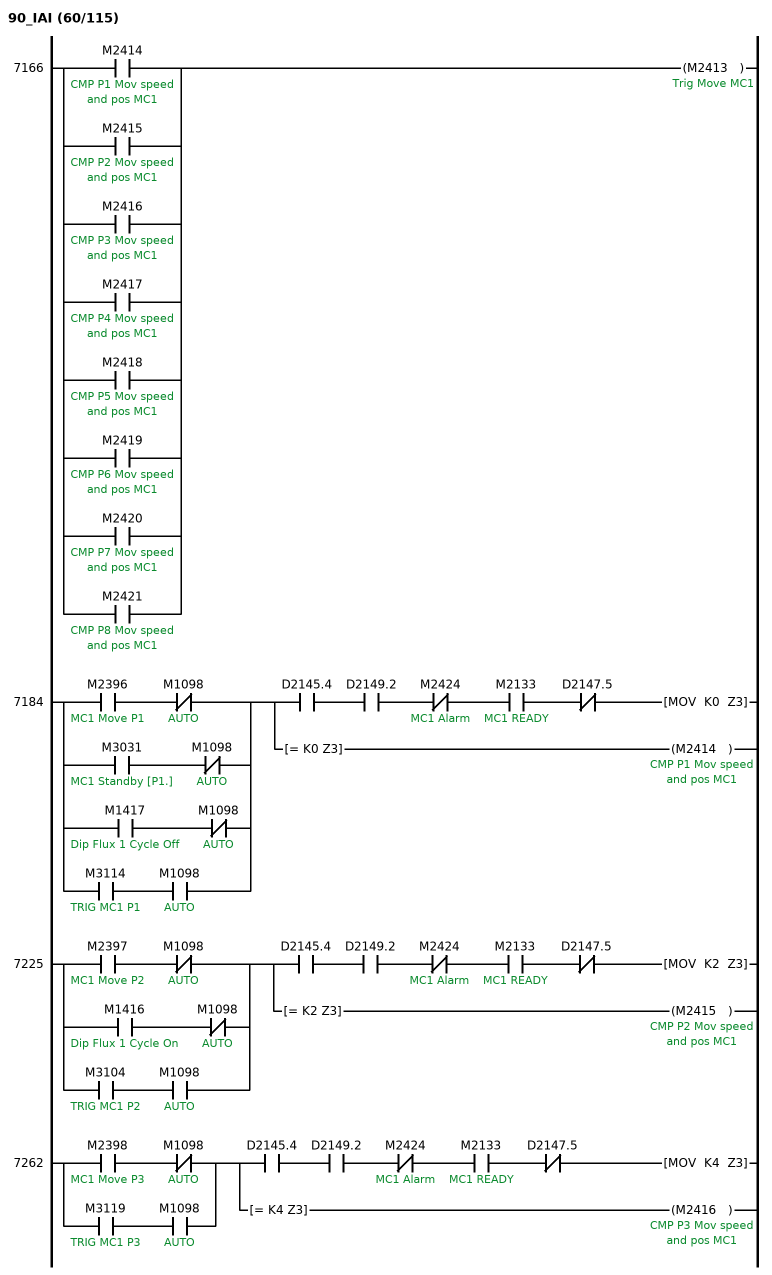
7166  LD      M2414  ; CMP P1 Mov speed and pos MC1
      OR      M2415  ; CMP P2 Mov speed and pos MC1
      OR      M2416  ; CMP P3 Mov speed and pos MC1
      OR      M2417  ; CMP P4 Mov speed and pos MC1
      OR      M2418  ; CMP P5 Mov speed and pos MC1
      OR      M2419  ; CMP P6 Mov speed and pos MC1
      OR      M2420  ; CMP P7 Mov speed and pos MC1
      OR      M2421  ; CMP P8 Mov speed and pos MC1
      OUT     M2413  ; Trig Move MC1
7184  LD      M2396  ; MC1 Move P1
      ANI     M1098  ; AUTO
      LD      M3031  ; MC1 Standby [P1.]
      ANI     M1098  ; AUTO
      ORB
      LD      M1417  ; Dip Flux 1 Cycle Off
      ANI     M1098  ; AUTO
      ORB
      LD      M3114  ; TRIG MC1 P1
      AND     M1098  ; AUTO
      ORB
      MPS
      AND     D2145.4
      AND     D2149.2
      ANI     M2424  ; MC1 Alarm
      AND     M2133  ; MC1 READY
      ANI     D2147.5
      MOV     K0 Z3
      MPP
      AND=    K0 Z3
      OUT     M2414  ; CMP P1 Mov speed and pos MC1
7225  LD      M2397  ; MC1 Move P2
      ANI     M1098  ; AUTO
      LD      M1416  ; Dip Flux 1 Cycle On
      ANI     M1098  ; AUTO
      ORB
      LD      M3104  ; TRIG MC1 P2
      AND     M1098  ; AUTO
      ORB
      MPS
      AND     D2145.4
      AND     D2149.2
      ANI     M2424  ; MC1 Alarm
      AND     M2133  ; MC1 READY
      ANI     D2147.5
      MOV     K2 Z3
      MPP
      AND=    K2 Z3
      OUT     M2415  ; CMP P2 Mov speed and pos MC1
7262  LD      M2398  ; MC1 Move P3
      ANI     M1098  ; AUTO
      LD      M3119  ; TRIG MC1 P3
      AND     M1098  ; AUTO
      ORB
      MPS
      AND     D2145.4
      AND     D2149.2
      ANI     M2424  ; MC1 Alarm
      AND     M2133  ; MC1 READY
      ANI     D2147.5
      MOV     K4 Z3
      MPP
      AND=    K4 Z3
      OUT     M2416  ; CMP P3 Mov speed and pos MC1
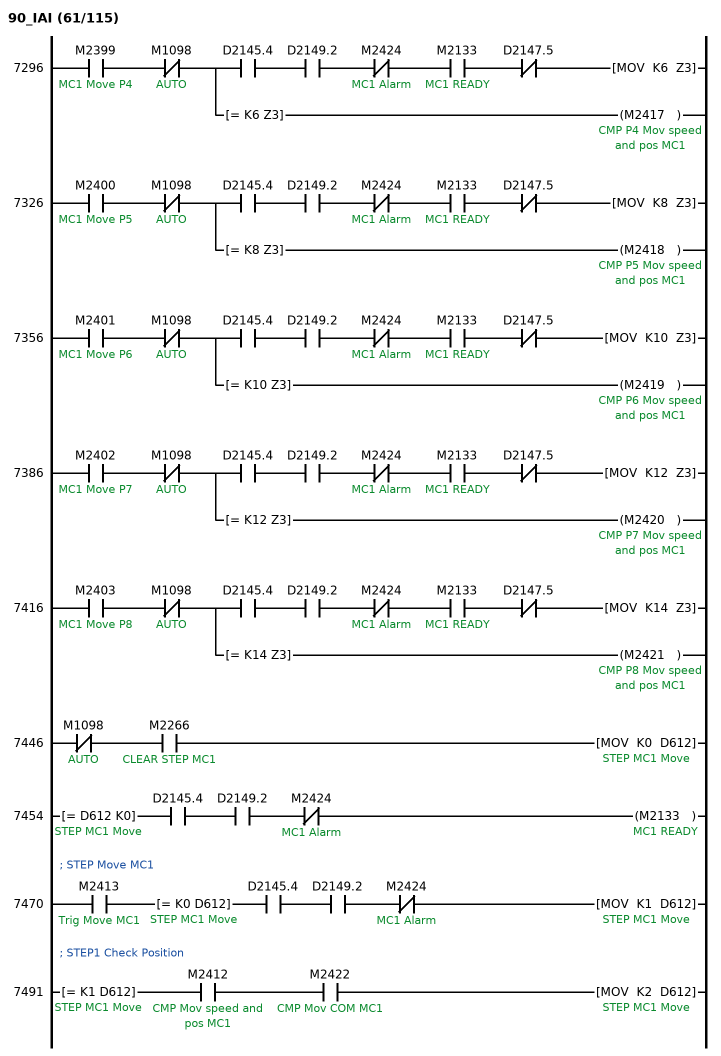
7296  LD      M2399  ; MC1 Move P4
      ANI     M1098  ; AUTO
      MPS
      AND     D2145.4
      AND     D2149.2
      ANI     M2424  ; MC1 Alarm
      AND     M2133  ; MC1 READY
      ANI     D2147.5
      MOV     K6 Z3
      MPP
      AND=    K6 Z3
      OUT     M2417  ; CMP P4 Mov speed and pos MC1
7326  LD      M2400  ; MC1 Move P5
      ANI     M1098  ; AUTO
      MPS
      AND     D2145.4
      AND     D2149.2
      ANI     M2424  ; MC1 Alarm
      AND     M2133  ; MC1 READY
      ANI     D2147.5
      MOV     K8 Z3
      MPP
      AND=    K8 Z3
      OUT     M2418  ; CMP P5 Mov speed and pos MC1
7356  LD      M2401  ; MC1 Move P6
      ANI     M1098  ; AUTO
      MPS
      AND     D2145.4
      AND     D2149.2
      ANI     M2424  ; MC1 Alarm
      AND     M2133  ; MC1 READY
      ANI     D2147.5
      MOV     K10 Z3
      MPP
      AND=    K10 Z3
      OUT     M2419  ; CMP P6 Mov speed and pos MC1
7386  LD      M2402  ; MC1 Move P7
      ANI     M1098  ; AUTO
      MPS
      AND     D2145.4
      AND     D2149.2
      ANI     M2424  ; MC1 Alarm
      AND     M2133  ; MC1 READY
      ANI     D2147.5
      MOV     K12 Z3
      MPP
      AND=    K12 Z3
      OUT     M2420  ; CMP P7 Mov speed and pos MC1
7416  LD      M2403  ; MC1 Move P8
      ANI     M1098  ; AUTO
      MPS
      AND     D2145.4
      AND     D2149.2
      ANI     M2424  ; MC1 Alarm
      AND     M2133  ; MC1 READY
      ANI     D2147.5
      MOV     K14 Z3
      MPP
      AND=    K14 Z3
      OUT     M2421  ; CMP P8 Mov speed and pos MC1
7446  LDI     M1098  ; AUTO
      AND     M2266  ; CLEAR STEP MC1
      MOV     K0 D612
7454  LD=     D612 K0  ; STEP MC1 Move
      AND     D2145.4
      AND     D2149.2
      ANI     M2424  ; MC1 Alarm
      OUT     M2133  ; MC1 READY
; STEP Move MC1
7470  LD      M2413  ; Trig Move MC1
      AND=    K0 D612  ; STEP MC1 Move
      AND     D2145.4
      AND     D2149.2
      ANI     M2424  ; MC1 Alarm
      MOV     K1 D612
; STEP1 Check Position
7491  LD=     K1 D612  ; STEP MC1 Move
      AND     M2412  ; CMP Mov speed and pos MC1
      AND     M2422  ; CMP Mov COM MC1
      MOV     K2 D612
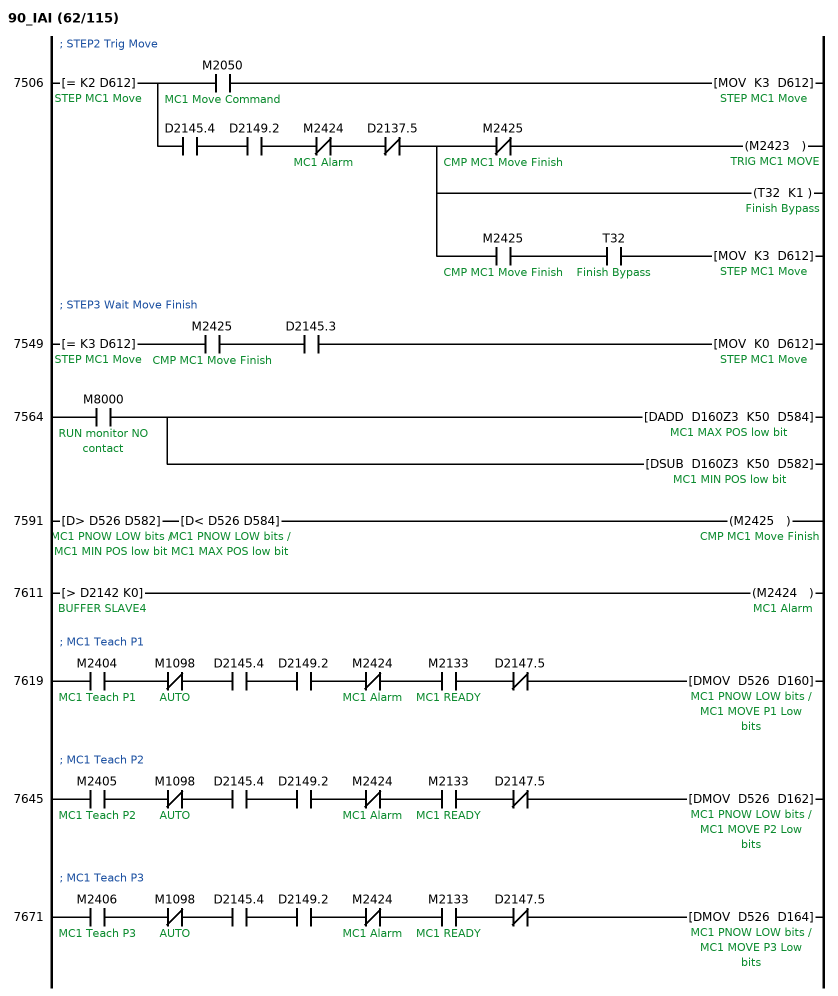
; STEP2 Trig Move
7506  LD=     K2 D612  ; STEP MC1 Move
      MPS
      AND     M2050  ; MC1 Move Command
      MOV     K3 D612
      MPP
      AND     D2145.4
      AND     D2149.2
      ANI     M2424  ; MC1 Alarm
      ANI     D2137.5
      MPS
      ANI     M2425  ; CMP MC1 Move Finish
      OUT     M2423  ; TRIG MC1 MOVE
      MPP
      OUT     T32 K1  ; Finish Bypass
      AND     M2425  ; CMP MC1 Move Finish
      AND     T32  ; Finish Bypass
      MOV     K3 D612
; STEP3 Wait Move Finish
7549  LD=     K3 D612  ; STEP MC1 Move
      AND     M2425  ; CMP MC1 Move Finish
      AND     D2145.3
      MOV     K0 D612
7564  LD      M8000  ; RUN monitor NO contact
      DADD    D160Z3 K50 D584  ; MC1 MAX POS low bit
      DSUB    D160Z3 K50 D582  ; MC1 MIN POS low bit
7591  LDD>    D526 D582  ; MC1 PNOW LOW bits / MC1 MIN POS low bit
      ANDD<   D526 D584  ; MC1 PNOW LOW bits / MC1 MAX POS low bit
      OUT     M2425  ; CMP MC1 Move Finish
7611  LD>     D2142 K0  ; BUFFER SLAVE4
      OUT     M2424  ; MC1 Alarm
; MC1 Teach P1
7619  LD      M2404  ; MC1 Teach P1
      ANI     M1098  ; AUTO
      AND     D2145.4
      AND     D2149.2
      ANI     M2424  ; MC1 Alarm
      AND     M2133  ; MC1 READY
      ANI     D2147.5
      DMOV    D526 D160  ; MC1 MOVE P1 Low bits
; MC1 Teach P2
7645  LD      M2405  ; MC1 Teach P2
      ANI     M1098  ; AUTO
      AND     D2145.4
      AND     D2149.2
      ANI     M2424  ; MC1 Alarm
      AND     M2133  ; MC1 READY
      ANI     D2147.5
      DMOV    D526 D162  ; MC1 MOVE P2 Low bits
; MC1 Teach P3
7671  LD      M2406  ; MC1 Teach P3
      ANI     M1098  ; AUTO
      AND     D2145.4
      AND     D2149.2
      ANI     M2424  ; MC1 Alarm
      AND     M2133  ; MC1 READY
      ANI     D2147.5
      DMOV    D526 D164  ; MC1 MOVE P3 Low bits
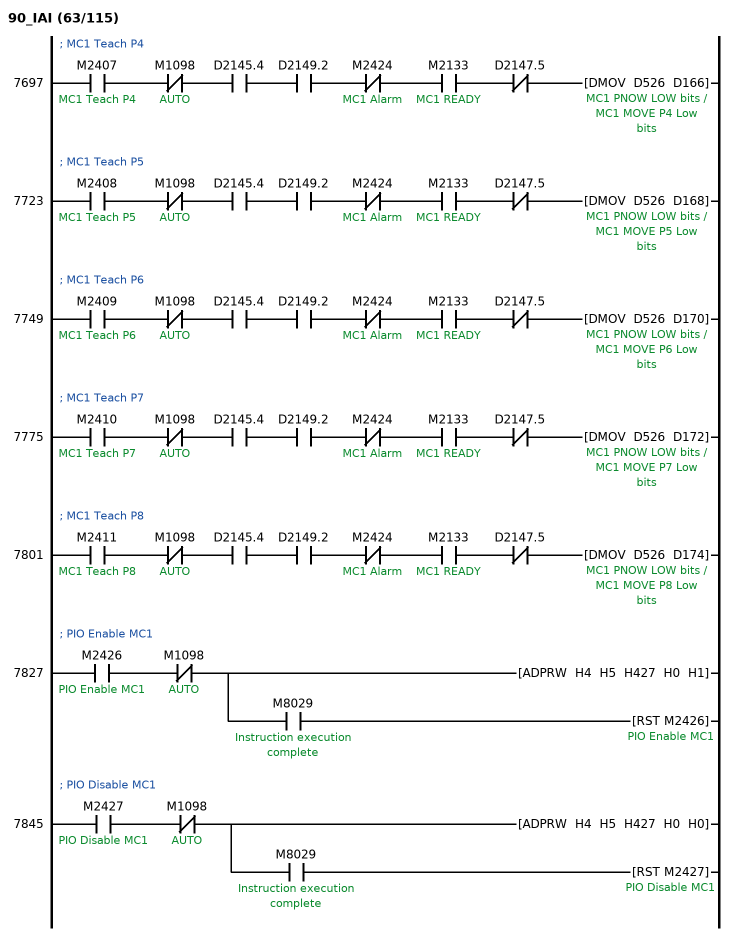
; MC1 Teach P4
7697  LD      M2407  ; MC1 Teach P4
      ANI     M1098  ; AUTO
      AND     D2145.4
      AND     D2149.2
      ANI     M2424  ; MC1 Alarm
      AND     M2133  ; MC1 READY
      ANI     D2147.5
      DMOV    D526 D166  ; MC1 MOVE P4 Low bits
; MC1 Teach P5
7723  LD      M2408  ; MC1 Teach P5
      ANI     M1098  ; AUTO
      AND     D2145.4
      AND     D2149.2
      ANI     M2424  ; MC1 Alarm
      AND     M2133  ; MC1 READY
      ANI     D2147.5
      DMOV    D526 D168  ; MC1 MOVE P5 Low bits
; MC1 Teach P6
7749  LD      M2409  ; MC1 Teach P6
      ANI     M1098  ; AUTO
      AND     D2145.4
      AND     D2149.2
      ANI     M2424  ; MC1 Alarm
      AND     M2133  ; MC1 READY
      ANI     D2147.5
      DMOV    D526 D170  ; MC1 MOVE P6 Low bits
; MC1 Teach P7
7775  LD      M2410  ; MC1 Teach P7
      ANI     M1098  ; AUTO
      AND     D2145.4
      AND     D2149.2
      ANI     M2424  ; MC1 Alarm
      AND     M2133  ; MC1 READY
      ANI     D2147.5
      DMOV    D526 D172  ; MC1 MOVE P7 Low bits
; MC1 Teach P8
7801  LD      M2411  ; MC1 Teach P8
      ANI     M1098  ; AUTO
      AND     D2145.4
      AND     D2149.2
      ANI     M2424  ; MC1 Alarm
      AND     M2133  ; MC1 READY
      ANI     D2147.5
      DMOV    D526 D174  ; MC1 MOVE P8 Low bits
; PIO Enable MC1
7827  LD      M2426  ; PIO Enable MC1
      ANI     M1098  ; AUTO
      ADPRW   H4 H5 H427 H0 H1
      AND     M8029  ; Instruction execution complete
      RST     M2426  ; PIO Enable MC1
; PIO Disable MC1
7845  LD      M2427  ; PIO Disable MC1
      ANI     M1098  ; AUTO
      ADPRW   H4 H5 H427 H0 H0
      AND     M8029  ; Instruction execution complete
      RST     M2427  ; PIO Disable MC1
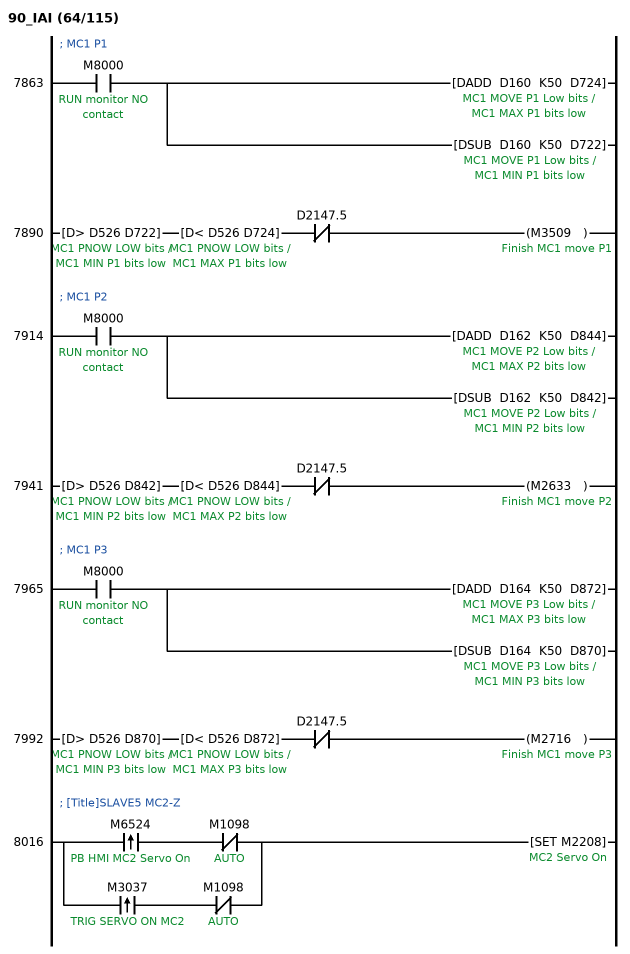
; MC1 P1
7863  LD      M8000  ; RUN monitor NO contact
      DADD    D160 K50 D724  ; MC1 MAX P1 bits low
      DSUB    D160 K50 D722  ; MC1 MIN P1 bits low
7890  LDD>    D526 D722  ; MC1 PNOW LOW bits / MC1 MIN P1 bits low
      ANDD<   D526 D724  ; MC1 PNOW LOW bits / MC1 MAX P1 bits low
      ANI     D2147.5
      OUT     M3509  ; Finish MC1 move P1
; MC1 P2
7914  LD      M8000  ; RUN monitor NO contact
      DADD    D162 K50 D844  ; MC1 MAX P2 bits low
      DSUB    D162 K50 D842  ; MC1 MIN P2 bits low
7941  LDD>    D526 D842  ; MC1 PNOW LOW bits / MC1 MIN P2 bits low
      ANDD<   D526 D844  ; MC1 PNOW LOW bits / MC1 MAX P2 bits low
      ANI     D2147.5
      OUT     M2633  ; Finish MC1 move P2
; MC1 P3
7965  LD      M8000  ; RUN monitor NO contact
      DADD    D164 K50 D872  ; MC1 MAX P3 bits low
      DSUB    D164 K50 D870  ; MC1 MIN P3 bits low
7992  LDD>    D526 D870  ; MC1 PNOW LOW bits / MC1 MIN P3 bits low
      ANDD<   D526 D872  ; MC1 PNOW LOW bits / MC1 MAX P3 bits low
      ANI     D2147.5
      OUT     M2716  ; Finish MC1 move P3
; [Title]SLAVE5 MC2-Z
8016  LDP     M6524  ; PB HMI MC2 Servo On
      ANI     M1098  ; AUTO
      LDP     M3037  ; TRIG SERVO ON MC2
      ANI     M1098  ; AUTO
      ORB
      SET     M2208  ; MC2 Servo On
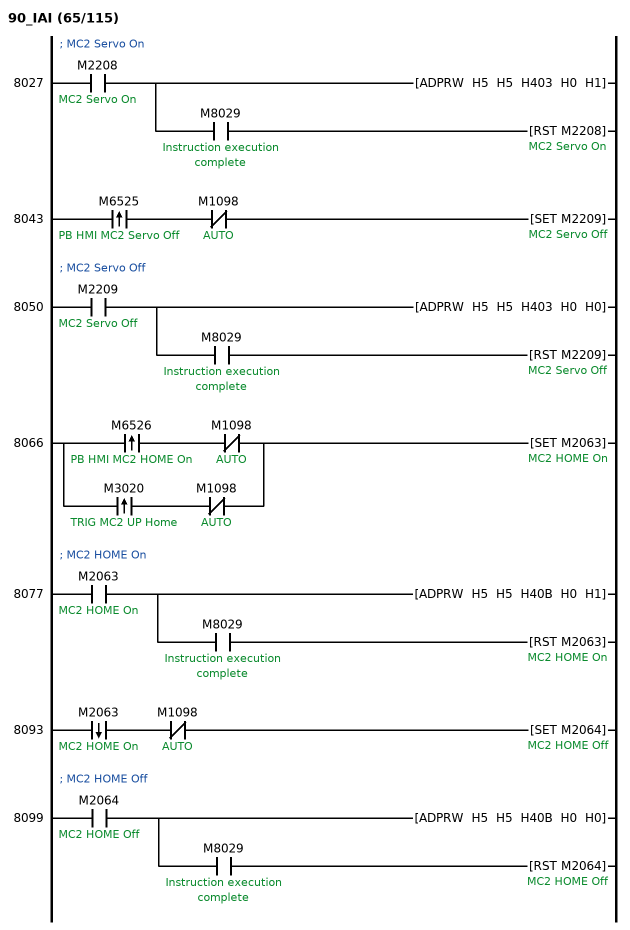
; MC2 Servo On
8027  LD      M2208  ; MC2 Servo On
      ADPRW   H5 H5 H403 H0 H1
      AND     M8029  ; Instruction execution complete
      RST     M2208  ; MC2 Servo On
8043  LDP     M6525  ; PB HMI MC2 Servo Off
      ANI     M1098  ; AUTO
      SET     M2209  ; MC2 Servo Off
; MC2 Servo Off
8050  LD      M2209  ; MC2 Servo Off
      ADPRW   H5 H5 H403 H0 H0
      AND     M8029  ; Instruction execution complete
      RST     M2209  ; MC2 Servo Off
8066  LDP     M6526  ; PB HMI MC2 HOME On
      ANI     M1098  ; AUTO
      LDP     M3020  ; TRIG MC2 UP Home
      ANI     M1098  ; AUTO
      ORB
      SET     M2063  ; MC2 HOME On
; MC2 HOME On
8077  LD      M2063  ; MC2 HOME On
      ADPRW   H5 H5 H40B H0 H1
      AND     M8029  ; Instruction execution complete
      RST     M2063  ; MC2 HOME On
8093  LDF     M2063  ; MC2 HOME On
      ANI     M1098  ; AUTO
      SET     M2064  ; MC2 HOME Off
; MC2 HOME Off
8099  LD      M2064  ; MC2 HOME Off
      ADPRW   H5 H5 H40B H0 H0
      AND     M8029  ; Instruction execution complete
      RST     M2064  ; MC2 HOME Off
